TYPE T_Wstring : WSTRING; END_TYPE

(* stored: Version 1.1.0.1
   DUT T_Wstring: Id {9dc87915-8ff7-4698-86bd-fc94d0da82fd} *)
